{attribute 'qualified_only'}
VAR_GLOBAL
	// Encoder reference values in counts = nm
	nYUP_ENC_REF : ULINT := 14760900;
	nYDWN_ENC_REF : ULINT := 13941900;
	nXUP_ENC_REF : ULINT := 24435400;
	nXDWN_ENC_REF : ULINT := 25239600;
END_VAR

(* stored: Version 1.1.0.1, ProductVersion 3.1.4022.12
   GVL GVL_M1L0: Id {623cea80-686b-4793-a8f5-8ca2e875142f} *)
